ABB RobotStudio station: JogRobot_20211110-155153.rsstn

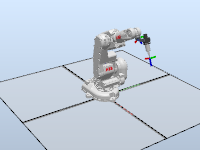
Station Basics1 (saved by RobotStudio 21.2.9526.0)
Controller CRB1100_4_47_Controller
  mechanical unit ROB_1: IRB140_6_81_C_03, 6 joints, base frame (0, 0, 0) mm
Layout (positions relative to the parent item):
  - IRB140_6_81_C_03 [mechanism, from Robots\IRB140_6_81_C_G_03.rslib] at (0, 0, 0) mm; joint values [0.0303, 0.1039, -0.5495, -0.0318, 0.9697, 0.0331] (rad or m)
  - MyTool [mechanism, from Training Objects\myTool.rslib] at (506.29, 13.63, 841.36) mm, rotated rx 180 ry 60 rz 180 deg
Attachment: MyTool is attached to IRB140_6_81_C_03 / Link6
Targets, tools, work objects and paths stored in the station, written as RAPID:
! task T_ROB1
MODULE CalibData
  PERS tooldata MyTool:=[TRUE,[[31.792631019,0,229.638935148],[0.945518576,0,0.325568154,0]],[1,[0,0,1],[1,0,0,0],0,0,0]];
ENDMODULE

